(* -----------------------------------------------------------------------------
| This sample has been supplied by Beckhoff As-Is and is intended only as an   |
| example implementation. Functionality is not guaranteed.                     |
----------------------------------------------------------------------------- *)

FUNCTION_BLOCK FB_VisuSim
VAR_INPUT
	bConveyor : BOOL;
	bWater : BOOL;
	bMint : BOOL;
	bCorkingRotation : BOOL;
	bCokingVertical : BOOL;
	bRefillWater : BOOL;
	bRefillMint : BOOL;
	bEmergencyButton : BOOL;
END_VAR
VAR_OUTPUT
	fPos : REAL;	
	bBottle : BOOL;
	nWaterLevel : INT;
	nMintLevel : INT;
	bCorkingRotationLimitSwitch : BOOL;
	bEmergency : BOOL;
END_VAR
VAR
	bInitialized : BOOL;	
	nCorkingRotationCnt : UINT;
	nCorkingRotationCntLowerLimit : UINT := 30;
	fbRefill : BLINK;
	fbRtRefill : R_TRIG;
END_VAR

(* -----------------------------------------------------------------------------
| This sample has been supplied by Beckhoff As-Is and is intended only as an   |
| example implementation. Functionality is not guaranteed.                     |
----------------------------------------------------------------------------- *)

IF NOT bInitialized THEN
	nWaterLevel := 32000;
	nMintLevel := 24000;
	bInitialized := TRUE;	
ELSE
	
	(* Simulazione pulsante di emergenza *)
	bEmergency := bEmergencyButton;	
	
	(* simulazione nastro trasportatore e sensore presenza bottiglia *)
	IF bConveyor THEN
		fPos := fPos + 0.1;
	END_IF
	
	IF fPos >= 120.0 THEN
		fPos := 0;
	END_IF
	
	bBottle := fPos >= 60.0 AND fPos <= 80.0;
	
	(* simulazione auto-approvvigionamento liquidi *) 
	fbRefill(ENABLE:= TRUE, TIMELOW:= T#15S, TIMEHIGH:= T#15S);
	fbRtRefill(CLK := fbRefill.OUT);
	IF fbRtRefill.Q THEN
		IF nWaterLevel < 11000 THEN
			bRefillWater := TRUE;
		END_IF
		IF nMintLevel < 9000 THEN
			bRefillMint := TRUE;
		END_IF
	END_IF
	
	(* simulazione livelli acqua e menta *)
	IF bWater THEN
		nWaterLevel := nWaterLevel - 11;
	END_IF
	
	IF nWaterLevel < 0 THEN
		nWaterLevel := 0;
	END_IF
	
	IF bRefillWater THEN
		nWaterLevel := nWaterLevel + 19567;
	END_IF
	
	IF bMint THEN
		nMintLevel := nMintLevel - 17;
	END_IF
	
	IF nMintLevel < 0 THEN
		nMintLevel := 0;
	END_IF
	
	IF bRefillMint THEN
		nMintLevel := nMintLevel + 20231;
	END_IF
	
	bRefillWater := FALSE;
	bRefillMint := FALSE;
	
	(* simulazione sensore tappatura *)
	IF bCokingVertical THEN
		IF bCorkingRotation THEN
			nCorkingRotationCnt := nCorkingRotationCnt + 1;
		END_IF
	ELSE
		nCorkingRotationCnt := 0;
	END_IF
	
	bCorkingRotationLimitSwitch := nCorkingRotationCnt > nCorkingRotationCntLowerLimit;
	
	
	
	
	
	
	
	
	
END_IF

END_FUNCTION_BLOCK

(* stored: Version 1.1.0.1, ProductVersion 3.1.4024.12
   POU FB_VisuSim: Id {3774dbef-c7d2-4a4d-811e-1fba5257b332}, SpecialFunc None *)
